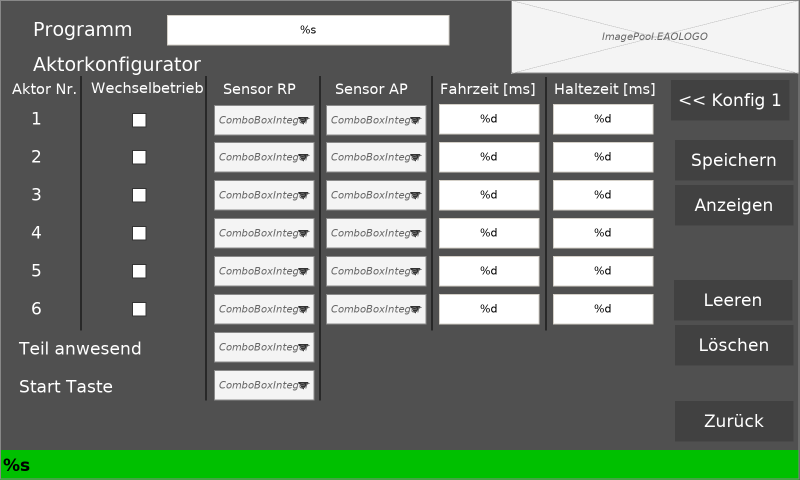
VISUALIZATION Konfig2  // 800x480
    Image (511,0 288x73), image: ImagePool.EAOLOGO
    Textfield (30,15 200x29), "Programm"
    Rectangle (0,450 799x30), "%s", text variable: MAIN.HMI.sStatus, colour variable: MAIN.HMI.nColorInfoBalken
        p3450524324: MAIN.HMI.nColorInfoBalken
    Textfield (220,74 109x30), "Sensor RP"
    Textfield (332,74 109x30), "Sensor AP"
    RoundedRectangle (675,325 118x40), "Löschen"
        OnMouseClick: execute { MAIN.HMI.bBtnProgrammLoeschen := TRUE; }
    Textfield (9,74 73x30), "Aktor Nr."
    Line (206,400) (206,76)
    Line (320,400) (320,76)
    Line (432,330) (432,76)
    Textfield (437,74 109x30), "Fahrzeit [ms]"
    Line (546,330) (546,77)
    Textfield (167,15 282x30), "%s", text variable: MAIN.HMI.ProgrammTemp.sName
        OnMouseClick: write the text variable via VisuDialogs.Keypad
    Textfield (551,74 109x30), "Haltezeit [ms]"
    RoundedRectangle (675,140 118x40), "Speichern", colour toggle: MAIN.fbWritePersistentData.BUSY
        OnMouseClick: execute { MAIN.HMI.bBtnProgrammSpeichern := TRUE; }
    RoundedRectangle (675,185 118x40), "Anzeigen"
        OnMouseClick: execute { MAIN.HMI.bBtnProgrammAnzeigen := TRUE; }
    Textfield (30,50 200x29), "Aktorkonfigurator"
    RoundedRectangle (671,80 118x40), "<< Konfig 1"
        OnMouseClick: change screen: Konfig1
    RoundedRectangle (2011,204 118x40), "<< Konfig 1", colour toggle: MAIN.fbWritePersistentData.BUSY
        OnMouseClick: execute { MAIN.HMI.bBtnProgrammSpeichern := TRUE; }
    Textfield (28,104 34x29), "1"
    Textfield (28,180 34x29), "3"
    Textfield (28,218 34x29), "4"
    Textfield (28,142 34x29), "2"
    Textfield (28,256 34x29), "5"
    Textfield (28,294 34x29), "6"
    Textfield (439,104 100x30), "%d", text variable: MAIN.HMI.ProgrammTemp.aAktorKonfig[1].nFahrZeit
        OnMouseClick: write the text variable via VisuDialogs.Numpad
    Textfield (553,104 100x30), "%d", text variable: MAIN.HMI.ProgrammTemp.aAktorKonfig[1].nHalteZeit
        OnMouseClick: write the text variable via VisuDialogs.Numpad
    Textfield (439,142 100x30), "%d", text variable: MAIN.HMI.ProgrammTemp.aAktorKonfig[2].nFahrZeit
        OnMouseClick: write the text variable via VisuDialogs.Numpad
    Textfield (553,142 100x30), "%d", text variable: MAIN.HMI.ProgrammTemp.aAktorKonfig[2].nHalteZeit
        OnMouseClick: write the text variable via VisuDialogs.Numpad
    Textfield (439,180 100x30), "%d", text variable: MAIN.HMI.ProgrammTemp.aAktorKonfig[3].nFahrZeit
        OnMouseClick: write the text variable via VisuDialogs.Numpad
    Textfield (553,180 100x30), "%d", text variable: MAIN.HMI.ProgrammTemp.aAktorKonfig[3].nHalteZeit
        OnMouseClick: write the text variable via VisuDialogs.Numpad
    Textfield (439,218 100x30), "%d", text variable: MAIN.HMI.ProgrammTemp.aAktorKonfig[4].nFahrZeit
        OnMouseClick: write the text variable via VisuDialogs.Numpad
    Textfield (553,218 100x30), "%d", text variable: MAIN.HMI.ProgrammTemp.aAktorKonfig[4].nHalteZeit
        OnMouseClick: write the text variable via VisuDialogs.Numpad
    Textfield (439,256 100x30), "%d", text variable: MAIN.HMI.ProgrammTemp.aAktorKonfig[5].nFahrZeit
        OnMouseClick: write the text variable via VisuDialogs.Numpad
    Textfield (553,256 100x30), "%d", text variable: MAIN.HMI.ProgrammTemp.aAktorKonfig[5].nHalteZeit
        OnMouseClick: write the text variable via VisuDialogs.Numpad
    Textfield (439,294 100x30), "%d", text variable: MAIN.HMI.ProgrammTemp.aAktorKonfig[6].nFahrZeit
        OnMouseClick: write the text variable via VisuDialogs.Numpad
    Textfield (553,294 100x30), "%d", text variable: MAIN.HMI.ProgrammTemp.aAktorKonfig[6].nHalteZeit
        OnMouseClick: write the text variable via VisuDialogs.Numpad
    ComboBoxInteger (214,105 100x30), variable: MAIN.HMI.ProgrammTemp.aAktorKonfig[1].nSensRuhePos
    ComboBoxInteger (326,105 100x30), variable: MAIN.HMI.ProgrammTemp.aAktorKonfig[1].nSensArbeitsPos
    Textfield (16,334 143x29), "Teil anwesend"
    ComboBoxInteger (214,332 100x30), variable: MAIN.HMI.ProgrammTemp.nTeilAnw
    ComboBoxInteger (214,142 100x30), variable: MAIN.HMI.ProgrammTemp.aAktorKonfig[2].nSensRuhePos
    ComboBoxInteger (326,142 100x30), variable: MAIN.HMI.ProgrammTemp.aAktorKonfig[2].nSensArbeitsPos
    ComboBoxInteger (214,180 100x30), variable: MAIN.HMI.ProgrammTemp.aAktorKonfig[3].nSensRuhePos
    ComboBoxInteger (326,180 100x30), variable: MAIN.HMI.ProgrammTemp.aAktorKonfig[3].nSensArbeitsPos
    ComboBoxInteger (214,218 100x30), variable: MAIN.HMI.ProgrammTemp.aAktorKonfig[4].nSensRuhePos
    ComboBoxInteger (326,218 100x30), variable: MAIN.HMI.ProgrammTemp.aAktorKonfig[4].nSensArbeitsPos
    ComboBoxInteger (214,256 100x30), variable: MAIN.HMI.ProgrammTemp.aAktorKonfig[5].nSensRuhePos
    ComboBoxInteger (326,256 100x30), variable: MAIN.HMI.ProgrammTemp.aAktorKonfig[5].nSensArbeitsPos
    ComboBoxInteger (214,294 100x30), variable: MAIN.HMI.ProgrammTemp.aAktorKonfig[6].nSensRuhePos
    ComboBoxInteger (326,294 100x30), variable: MAIN.HMI.ProgrammTemp.aAktorKonfig[6].nSensArbeitsPos
    Textfield (16,372 143x29), "Start Taste"
    ComboBoxInteger (214,370 100x30), variable: MAIN.HMI.ProgrammTemp.nFussschalterAktiv, text list: 'TL_JaNein'
    Checkbox (130,105 32x30), variable: MAIN.HMI.ProgrammTemp.aAktorKonfig[1].bReversierBetrieb
    RoundedRectangle (675,401 118x40), "Zurück"
        OnMouseClick: change screen: Zyklusbetrieb
    RoundedRectangle (674,280 118x40), "Leeren"
        OnMouseClick: execute { MAIN.HMI.bBtnKonfigLeeren := TRUE; }
    Checkbox (130,142 32x30), variable: MAIN.HMI.ProgrammTemp.aAktorKonfig[2].bReversierBetrieb
    Checkbox (130,180 32x30), variable: MAIN.HMI.ProgrammTemp.aAktorKonfig[3].bReversierBetrieb
    Checkbox (130,218 32x30), variable: MAIN.HMI.ProgrammTemp.aAktorKonfig[4].bReversierBetrieb
    Checkbox (130,256 32x30), variable: MAIN.HMI.ProgrammTemp.aAktorKonfig[5].bReversierBetrieb
    Checkbox (130,294 32x30), variable: MAIN.HMI.ProgrammTemp.aAktorKonfig[6].bReversierBetrieb
    Textfield (88,73 120x30), "Wechselbetrieb"
    Line (81,330) (81,76)
    Group (826,90 645x290)
        p3560616238: MAIN.HMI.nPopUpXOffset
        RoundedRectangle (0,0 645x290), "%s", text variable: MAIN.HMI.sPopUpText, colour toggle: MAIN.fbWritePersistentData.BUSY, invisible if: NOT MAIN.HMI.bPopUpAnzeigen
        RoundedRectangle (128,197 118x40), "Ja", colour toggle: MAIN.fbWritePersistentData.BUSY, invisible if: NOT MAIN.HMI.bPopUpAnzeigen
            OnMouseClick: execute { MAIN.HMI.bBtnPopUpJa := TRUE; }
        RoundedRectangle (405,198 118x40), "Nein", colour toggle: MAIN.fbWritePersistentData.BUSY, invisible if: NOT MAIN.HMI.bPopUpAnzeigen
            OnMouseClick: execute { MAIN.HMI.bBtnPopUpNein := TRUE; }
END_VISUALIZATION

(* stored: Version 1.1.0.1, ProductVersion 3.1.4024.12
   Visu Konfig2: Id {81accf57-12e0-4a13-ab42-3ff4182b71fa} *)
